{attribute 'enable_dynamic_creation'}
FUNCTION_BLOCK Station IMPLEMENTS ITF_Cyclic, ITF_Station
VAR
	MyTrackPosition : LREAL;
END_VAR

{warning 'add method implementation '}
METHOD Cycle : BOOL
END_METHOD

METHOD Position : BOOL
VAR_INPUT
	StationPosition	: LREAL;
END_VAR
MyTrackPosition := StationPosition;
END_METHOD

END_FUNCTION_BLOCK

(* stored: Version 1.1.0.1, ProductVersion 3.1.4024.12
   POU Station: Id {3a164f31-1435-4c24-a4b9-f33358c56274}, SpecialFunc None
   Method Cycle: Id {4d5d8ab9-24a7-46b5-9b8b-8d304d0099b1}
   Method Position: Id {6213e8a0-7312-49ca-b711-7cdb926089fa} *)
